DATA_BLOCK "GeneralDebug"
VAR
  Debug : Array[1..99] of Bool;
END_VAR
BEGIN
END_DATA_BLOCK
